// TIA Portal project "Test Buttom Color" (V16)

(* hardware
DEVICE "HMI_1"  TP1200 Comfort Portrait
   slot 0: "HMI_1"  TP1200 Comfort Portrait  6AV2 124-0MC01-0AX0  16.0.0.0
   slot 1: "HMI_RT_1"  TP1200 Comfort Portrait  6AV2 124-0MC01-0AX0  16.0.0.0
   slot 5: "HMI_1.IE_CP_1"  PROFINET Interface  16.0.0.0
      slot 1: "PROFINET Interface_1"  PROFINET Interface
         slot 1: "Port_1"  Port
         slot 2: "Port_2"  Port
   slot 7: "HMI_1.MPI/DP_CP_1"  MPI/DP Interface  16.0.0.0
DEVICE "S7-1200 station_1"  S7-1200 Station
   slot 0: "Rack_0"  S7-1200 Rack  Rack  V1.0
   slot 1: "PLC_1"  CPU 1214C DC/DC/Rly  6ES7 214-1HG40-0XB0  V4.4
*)

// ===== PLC "PLC_1"  CPU 1214C DC/DC/Rly =====

DATA_BLOCK "Test"   // DB1
{ S7_Optimized_Access := 'TRUE' }
VERSION : 0.1
   VAR
      Start : Bool;
      Stop : Bool;
   END_VAR
BEGIN
END_DATA_BLOCK

ORGANIZATION_BLOCK "Main"   // OB1, LAD, ProgramCycle
TITLE = "Main Program Sweep (Cycle)"
{ S7_Optimized_Access := 'TRUE' }
VERSION : 0.1
   VAR_INPUT
      Initial_Call : Bool;   // Initial call of this OB
      Remanence : Bool;   // =True, if remanent data are available
   END_VAR
BEGIN
END_ORGANIZATION_BLOCK

(* ===== HMI "HMI_RT_1" =====
system functions are stored by id; their names below are inferred from use
connection "HMI_Connection_1": ETHERNET, S7_1200_OMS

HMI tags "Default tag table"
   "Start" : Bool = PLC Test.Start, 1 s
   "Stop" : Bool = PLC Test.Stop, 1 s

screen "Screen_1" 800x1280
   Button "Button_1" at 286,138 size 96x32; TextOff 'START'
      on Click: SetBit("Start")
      Appearance <- "Start"
   Button "Button_2" at 458,133 size 96x32; TextOff 'STOP'
      on Click: SetBit("Stop")
      Appearance <- "Stop"
*)